// TIA Portal V17 export
// export: Created 2022-07-28T18:02:47.3020839Z, ExportSetting None, DisplayName Totally Integrated Automation Portal, DisplayVersion V17, DisplayName TIA Portal Openness, DisplayVersion V17, DisplayName TIA Portal Teamcenter Gateway, DisplayVersion V17, DisplayName TIA Portal Version Control Interface, DisplayVersion V17, DisplayName TIA Portal Test Suite Advanced, DisplayVersion V17, DisplayName SINAMICS Startdrive Advanced, DisplayVersion V17, DisplayName SINAMICS DCC, DisplayVersion V17, DisplayName SINAMICS Startdrive G130, G150, S120, S150, SINAMICS MV, S210, DisplayVersion V17, DisplayName SINAMICS Startdrive G110M, G120, G120C, G120D, G120P, G115D, DisplayVersion V17, DisplayName STEP 7 Professional, DisplayVersion V17, DisplayName SIMATIC Energy Suite, DisplayVersion V17, DisplayName STEP 7 CFC, DisplayVersion V17, DisplayName STEP 7 Safety, DisplayVersion V17, DisplayName WinCC Advanced / Unified PC, DisplayVersion V17, DisplayName SIMATIC Visualization Architect, DisplayVersion V17
FUNCTION_BLOCK "Internal_H05_FB"   // FB11, SCL
TITLE = InternalH01
{ S7_Optimized_Access := 'TRUE' }
// Proccess signals from fuses, safety and others internal devices
// stored: MemoryReserve 100, SetENOAutomatically false
   VAR_INPUT
      I_CmdGeneralReset { ExternalAccessible := 'False'; ExternalVisible := 'False'; ExternalWritable := 'False'} : Bool;   // 0 ⮥ 1 = Input general reset ERROR/Interlocks
      IR_CycleTime { ExternalAccessible := 'False'; ExternalVisible := 'False'; ExternalWritable := 'False'} : Real := 0.0;   // Time of last PLC cycle, sec
      I_Initialization { ExternalAccessible := 'False'; ExternalVisible := 'False'; ExternalWritable := 'False'} : Bool := FALSE;   // 1 = Restart PLC is active (First scan)
      I_One_1s { ExternalAccessible := 'False'; ExternalVisible := 'False'; ExternalWritable := 'False'} : Bool;   // 1 = One cycle per one seccond pulse
      I_Sup24_Ok { ExternalAccessible := 'False'; ExternalVisible := 'False'; ExternalWritable := 'False'} : Bool;   // 24 VDC OK 004 -T1
      I_UPS_Alarm_Ok { ExternalAccessible := 'False'; ExternalVisible := 'False'; ExternalWritable := 'False'} : Bool;   // БЛОК безперебійного електроживлення ALARM 004 -K1.1
      I_UPS_Bat_Ok { ExternalAccessible := 'False'; ExternalVisible := 'False'; ExternalWritable := 'False'} : Bool;   // БЛОК безперебійного електроживлення BAT. 004 -K1.2
      I_QF_DQ_Ok { ExternalAccessible := 'False'; ExternalVisible := 'False'; ExternalWritable := 'False'} : Bool;   // Живлення модулів DO 004 -F4
      I_QF_AI_Ok { ExternalAccessible := 'False'; ExternalVisible := 'False'; ExternalWritable := 'False'} : Bool;   // Живлення модулів АІ 004 -F5
      I_QF_AQ_Ok { ExternalAccessible := 'False'; ExternalVisible := 'False'; ExternalWritable := 'False'} : Bool;   // Живлення модулів АО 004 -F6
      I_QF_Desmet_IM_Ok { ExternalAccessible := 'False'; ExternalVisible := 'False'; ExternalWritable := 'False'} : Bool;   // Живлення ЕТ станції для контролера DESMET 004 -F7
      I_QF_Desmet_DI_DQ_Ok { ExternalAccessible := 'False'; ExternalVisible := 'False'; ExternalWritable := 'False'} : Bool;   // Жилвення модулів DI та DO для контролера DESMET 004 -F8
      I_QF_Desmet_AI_AQ_Ok { ExternalAccessible := 'False'; ExternalVisible := 'False'; ExternalWritable := 'False'} : Bool;   // Живлення модулів AI та АO для контролера DESMET 004 -F9
      I_QF_Inv_Ctrl_Ok { ExternalAccessible := 'False'; ExternalVisible := 'False'; ExternalWritable := 'False'} : Bool;   // Живлення модулів керування частотників 004 -F10
      I_QF_Inv_STO_Ok { ExternalAccessible := 'False'; ExternalVisible := 'False'; ExternalWritable := 'False'} : Bool;   // Живлення STO контактів, частотних перетворювачів 004 -F11
      I_QF_Internal_Ok { ExternalAccessible := 'False'; ExternalVisible := 'False'; ExternalWritable := 'False'} : Bool;   // Живлення внутрішніх кіл 004 -F12
      I_QF_SafRelay_Ok { ExternalAccessible := 'False'; ExternalVisible := 'False'; ExternalWritable := 'False'} : Bool;   // Живлення реле безпеки 004 -F13
      I_QF_Analog_Ok { ExternalAccessible := 'False'; ExternalVisible := 'False'; ExternalWritable := 'False'} : Bool;   // Живлення аналогових сигналів 004 -F14
      I_QF_ThermoRelay_Ok { ExternalAccessible := 'False'; ExternalVisible := 'False'; ExternalWritable := 'False'} : Bool;   // Живлення термореле 004 -F15
      I_QF_VlvDisFoam_Ok { ExternalAccessible := 'False'; ExternalVisible := 'False'; ExternalWritable := 'False'} : Bool;   // Живлення клапанів ємності антивспінювача 004 -F16
      I_QF_FlowMeters_Ok { ExternalAccessible := 'False'; ExternalVisible := 'False'; ExternalWritable := 'False'} : Bool;   // Живлення витратомірів 004 -F17
      I_QF_VlvVitamin_Ok { ExternalAccessible := 'False'; ExternalVisible := 'False'; ExternalWritable := 'False'} : Bool;   // Живлення клапанів ємності вітамінів 004 -F18
      I_QF_DI_DQ_1_Ok { ExternalAccessible := 'False'; ExternalVisible := 'False'; ExternalWritable := 'False'} : Bool;   // Живлення дискретних сигналів 004 -F19
      I_QF_DI_DQ_2_Ok { ExternalAccessible := 'False'; ExternalVisible := 'False'; ExternalWritable := 'False'} : Bool;   // Живлення дискретних сигналів 004 -F20
      I_QS_Scalance_Ok { ExternalAccessible := 'False'; ExternalVisible := 'False'; ExternalWritable := 'False'} : Bool;   // Живлення скаланса 004 -F21
      I_SB_ES_Box_Ok { ExternalAccessible := 'False'; ExternalVisible := 'False'; ExternalWritable := 'False'} : Bool;   // Аварійний стоп 005 -SB1
      I_SB_ES_Ack_Ok { ExternalAccessible := 'False'; ExternalVisible := 'False'; ExternalWritable := 'False'} : Bool;   // Квітування 005 -SB2
      I_KM_SafRelay_Ok { ExternalAccessible := 'False'; ExternalVisible := 'False'; ExternalWritable := 'False'} : Bool;   // Доп. котакти контакторів кіл безпеки 005 -KM2
   END_VAR
   VAR_OUTPUT
      QW_STW { ExternalWritable := 'False'} : Word;   // Status for HMI
      QW_MW1 { ExternalWritable := 'False'} : Word;   // Message word for HMI 1
      QW_MW2 { ExternalWritable := 'False'} : Word := 16#0;   // Message word for HMI 2
      QW_MW3 { ExternalWritable := 'False'} : Word := 16#0;   // Message word for HMI 3
      Q_Reset { ExternalAccessible := 'False'; ExternalVisible := 'False'; ExternalWritable := 'False'} : Bool;   // 1 = Reset external err
      Q_SomeErr { ExternalAccessible := 'False'; ExternalVisible := 'False'; ExternalWritable := 'False'} : Bool;   // 1 = Some err occured
      Q_Sup24_Ok { ExternalAccessible := 'False'; ExternalVisible := 'False'; ExternalWritable := 'False'} : Bool;   // 24 VDC OK 004 -T1
      Q_UPS_Alarm_Ok { ExternalAccessible := 'False'; ExternalVisible := 'False'; ExternalWritable := 'False'} : Bool;   // БЛОК безперебійного електроживлення ALARM 004 -K1.1
      Q_UPS_Bat_Ok { ExternalAccessible := 'False'; ExternalVisible := 'False'; ExternalWritable := 'False'} : Bool;   // БЛОК безперебійного електроживлення BAT. 004 -K1.2
      Q_QF_DQ_Ok { ExternalAccessible := 'False'; ExternalVisible := 'False'; ExternalWritable := 'False'} : Bool;   // Живлення модулів DO 004 -F4
      Q_QF_AI_Ok { ExternalAccessible := 'False'; ExternalVisible := 'False'; ExternalWritable := 'False'} : Bool;   // Живлення модулів АІ 004 -F5
      Q_QF_AQ_Ok { ExternalAccessible := 'False'; ExternalVisible := 'False'; ExternalWritable := 'False'} : Bool;   // Живлення модулів АО 004 -F6
      Q_QF_Desmet_IM_Ok { ExternalAccessible := 'False'; ExternalVisible := 'False'; ExternalWritable := 'False'} : Bool;   // Живлення ЕТ станції для контролера DESMET 004 -F7
      Q_QF_Desmet_DI_DQ_Ok { ExternalAccessible := 'False'; ExternalVisible := 'False'; ExternalWritable := 'False'} : Bool;   // Жилвення модулів DI та DO для контролера DESMET 004 -F8
      Q_QF_Desmet_AI_AQ_Ok { ExternalAccessible := 'False'; ExternalVisible := 'False'; ExternalWritable := 'False'} : Bool;   // Живлення модулів AI та АO для контролера DESMET 004 -F9
      Q_QF_Inv_Ctrl_Ok { ExternalAccessible := 'False'; ExternalVisible := 'False'; ExternalWritable := 'False'} : Bool;   // Живлення модулів керування частотників 004 -F10
      Q_QF_Inv_STO_Ok { ExternalAccessible := 'False'; ExternalVisible := 'False'; ExternalWritable := 'False'} : Bool;   // Живлення STO контактів, частотних перетворювачів 004 -F11
      Q_QF_Internal_Ok { ExternalAccessible := 'False'; ExternalVisible := 'False'; ExternalWritable := 'False'} : Bool;   // Живлення внутрішніх кіл 004 -F12
      Q_QF_SafRelay_Ok { ExternalAccessible := 'False'; ExternalVisible := 'False'; ExternalWritable := 'False'} : Bool;   // Живлення реле безпеки 004 -F13
      Q_QF_Analog_Ok { ExternalAccessible := 'False'; ExternalVisible := 'False'; ExternalWritable := 'False'} : Bool;   // Живлення аналогових сигналів 004 -F14
      Q_QF_ThermoRelay_Ok { ExternalAccessible := 'False'; ExternalVisible := 'False'; ExternalWritable := 'False'} : Bool;   // Живлення термореле 004 -F15
      Q_QF_VlvDisFoam_Ok { ExternalAccessible := 'False'; ExternalVisible := 'False'; ExternalWritable := 'False'} : Bool;   // Живлення клапанів ємності антивспінювача 004 -F16
      Q_QF_FlowMeters_Ok { ExternalAccessible := 'False'; ExternalVisible := 'False'; ExternalWritable := 'False'} : Bool;   // Живлення витратомірів 004 -F17
      Q_QF_VlvVitamin_Ok { ExternalAccessible := 'False'; ExternalVisible := 'False'; ExternalWritable := 'False'} : Bool;   // Живлення клапанів ємності вітамінів 004 -F18
      Q_QF_DI_DQ_1_Ok { ExternalAccessible := 'False'; ExternalVisible := 'False'; ExternalWritable := 'False'} : Bool;   // Живлення дискретних сигналів 004 -F19
      Q_QF_DI_DQ_2_Ok { ExternalAccessible := 'False'; ExternalVisible := 'False'; ExternalWritable := 'False'} : Bool;   // Живлення дискретних сигналів 004 -F20
      Q_QS_Scalance_Ok { ExternalAccessible := 'False'; ExternalVisible := 'False'; ExternalWritable := 'False'} : Bool;   // Живлення скаланса 004 -F21
      Q_KM_SafRelay_Ok { ExternalAccessible := 'False'; ExternalVisible := 'False'; ExternalWritable := 'False'} : Bool;   // Доп. котакти контакторів кіл безпеки 005 -KM2
   END_VAR
   VAR_IN_OUT
      II_CMD : Int;   // Command from HMI for current box
   END_VAR
   VAR
      s_Sup24_Err { ExternalAccessible := 'False'; ExternalVisible := 'False'; ExternalWritable := 'False'} : Bool;   // 24 VDC OK 004 -T1
      s_UPS_Alarm_Err { ExternalAccessible := 'False'; ExternalVisible := 'False'; ExternalWritable := 'False'} : Bool;   // БЛОК безперебійного електроживлення ALARM 004 -K1.1
      s_UPS_Bat_Err { ExternalAccessible := 'False'; ExternalVisible := 'False'; ExternalWritable := 'False'} : Bool;   // БЛОК безперебійного електроживлення BAT. 004 -K1.2
      s_QF_DQ_Err { ExternalAccessible := 'False'; ExternalVisible := 'False'; ExternalWritable := 'False'} : Bool;   // Живлення модулів DO 004 -F4
      s_QF_AI_Err { ExternalAccessible := 'False'; ExternalVisible := 'False'; ExternalWritable := 'False'} : Bool;   // Живлення модулів АІ 004 -F5
      s_QF_AQ_Err { ExternalAccessible := 'False'; ExternalVisible := 'False'; ExternalWritable := 'False'} : Bool;   // Живлення модулів АО 004 -F6
      s_QF_Desmet_IM_Err { ExternalAccessible := 'False'; ExternalVisible := 'False'; ExternalWritable := 'False'} : Bool;   // Живлення ЕТ станції для контролера DESMET 004 -F7
      s_QF_Desmet_DI_DQ_Err { ExternalAccessible := 'False'; ExternalVisible := 'False'; ExternalWritable := 'False'} : Bool;   // Жилвення модулів DI та DO для контролера DESMET 004 -F8
      s_QF_Desmet_AI_AQ_Err { ExternalAccessible := 'False'; ExternalVisible := 'False'; ExternalWritable := 'False'} : Bool;   // Живлення модулів AI та АO для контролера DESMET 004 -F9
      s_QF_Inv_Ctrl_Err { ExternalAccessible := 'False'; ExternalVisible := 'False'; ExternalWritable := 'False'} : Bool;   // Живлення модулів керування частотників 004 -F10
      s_QF_Inv_STO_Err { ExternalAccessible := 'False'; ExternalVisible := 'False'; ExternalWritable := 'False'} : Bool;   // Живлення STO контактів, частотних перетворювачів 004 -F11
      s_QF_Internal_Err { ExternalAccessible := 'False'; ExternalVisible := 'False'; ExternalWritable := 'False'} : Bool;   // Живлення внутрішніх кіл 004 -F12
      s_QF_SafRelay_Err { ExternalAccessible := 'False'; ExternalVisible := 'False'; ExternalWritable := 'False'} : Bool;   // Живлення реле безпеки 004 -F13
      s_QF_Analog_Err { ExternalAccessible := 'False'; ExternalVisible := 'False'; ExternalWritable := 'False'} : Bool;   // Живлення аналогових сигналів 004 -F14
      s_QF_ThermoRelay_Err { ExternalAccessible := 'False'; ExternalVisible := 'False'; ExternalWritable := 'False'} : Bool;   // Живлення термореле 004 -F15
      s_QF_VlvDisFoam_Err { ExternalAccessible := 'False'; ExternalVisible := 'False'; ExternalWritable := 'False'} : Bool;   // Живлення клапанів ємності антивспінювача 004 -F16
      s_QF_FlowMeters_Err { ExternalAccessible := 'False'; ExternalVisible := 'False'; ExternalWritable := 'False'} : Bool;   // Живлення витратомірів 004 -F17
      s_QF_VlvVitamin_Err { ExternalAccessible := 'False'; ExternalVisible := 'False'; ExternalWritable := 'False'} : Bool;   // Живлення клапанів ємності вітамінів 004 -F18
      s_QF_DI_DQ_1_Err { ExternalAccessible := 'False'; ExternalVisible := 'False'; ExternalWritable := 'False'} : Bool;   // Живлення дискретних сигналів 004 -F19
      s_QF_DI_DQ_2_Err { ExternalAccessible := 'False'; ExternalVisible := 'False'; ExternalWritable := 'False'} : Bool;   // Живлення дискретних сигналів 004 -F20
      s_QS_Scalance_Err { ExternalAccessible := 'False'; ExternalVisible := 'False'; ExternalWritable := 'False'} : Bool;   // Живлення скаланса 004 -F21
      s_KM_SafRelay_Err { ExternalAccessible := 'False'; ExternalVisible := 'False'; ExternalWritable := 'False'} : Bool;   // Доп. котакти контакторів кіл безпеки 005 -KM2
      s_TP_Reset { ExternalAccessible := 'False'; ExternalVisible := 'False'; ExternalWritable := 'False'} : "Lib_FB_Timer_TP_Simple";
   END_VAR
   VAR_TEMP
      t_ResetHMI : Bool;   // Reset from HMI
      t_ResetLogic : Bool;   // Reset for logic
      t_SomeErr : Bool;   // 1 = Some err occured
      ti_LogicCMD : Int;   // CMD for logic
      tw_STW : Word;   // Status for HMI
      tw_MW1 : Word;   // Message word for HMI 1
      tw_MW2 : Word;   // Message word for HMI 2
      tw_MW3 : Word;   // Message word for HMI 3
   END_VAR
BEGIN
   REGION Initialization
       IF #II_CMD <> 0
       THEN
           #ti_LogicCMD := #II_CMD;
           #II_CMD := 0;
       ELSE
           #ti_LogicCMD := 0;
       END_IF;

       #t_ResetHMI := false;
       #tw_STW := w#16#0;
       #tw_MW1 := w#16#0;
       #tw_MW2 := w#16#0;
       #tw_MW3 := w#16#0;
   END_REGION

   REGION Reset for logic
       //Reset from HMI
       CASE #ti_LogicCMD OF
           31..32:  //Reset
               #t_ResetHMI := true;
           ELSE  // Statement section ELSE
               ;
       END_CASE;

       //Reset for logic
       #t_ResetLogic := #t_ResetHMI
       OR #I_CmdGeneralReset
       OR #I_SB_ES_Ack_Ok;

       #s_TP_Reset(IR_CycleTime:=#IR_CycleTime,
                   IB_StartTimerInput:=#t_ResetLogic,
                   IR_SpTime:=2.0,
                   QB_TimerOut=>#t_ResetLogic);

   END_REGION

   REGION Catch errors
       #s_Sup24_Err := (NOT #I_Sup24_Ok
       OR (#s_Sup24_Err
       AND NOT #t_ResetLogic))
       AND NOT #I_Initialization;

       #s_UPS_Alarm_Err := (NOT #I_UPS_Alarm_Ok
       OR (#s_UPS_Alarm_Err
       AND NOT #t_ResetLogic))
       AND NOT #I_Initialization;

       #s_UPS_Bat_Err := (NOT #I_UPS_Bat_Ok
       OR (#s_UPS_Bat_Err
       AND NOT #t_ResetLogic))
       AND NOT #I_Initialization;

       #s_QF_DQ_Err := (NOT #I_QF_DQ_Ok
       OR (#s_QF_DQ_Err
       AND NOT #t_ResetLogic))
       AND NOT #I_Initialization;

       #s_QF_AI_Err := (NOT #I_QF_AI_Ok
       OR (#s_QF_AI_Err
       AND NOT #t_ResetLogic))
       AND NOT #I_Initialization;

       #s_QF_AQ_Err := (NOT #I_QF_AQ_Ok
       OR (#s_QF_AQ_Err
       AND NOT #t_ResetLogic))
       AND NOT #I_Initialization;

       #s_QF_Desmet_IM_Err := (NOT #I_QF_Desmet_IM_Ok
       OR (#s_QF_Desmet_IM_Err
       AND NOT #t_ResetLogic))
       AND NOT #I_Initialization;

       #s_QF_Desmet_DI_DQ_Err := (NOT #I_QF_Desmet_DI_DQ_Ok
       OR (#s_QF_Desmet_DI_DQ_Err
       AND NOT #t_ResetLogic))
       AND NOT #I_Initialization;

       #s_QF_Desmet_AI_AQ_Err := (NOT #I_QF_Desmet_AI_AQ_Ok
       OR (#s_QF_Desmet_AI_AQ_Err
       AND NOT #t_ResetLogic))
       AND NOT #I_Initialization;

       #s_QF_Inv_Ctrl_Err := (NOT #I_QF_Inv_Ctrl_Ok
       OR (#s_QF_Inv_Ctrl_Err
       AND NOT #t_ResetLogic))
       AND NOT #I_Initialization;

       #s_QF_Inv_STO_Err := (NOT #I_QF_Inv_STO_Ok
       OR (#s_QF_Inv_STO_Err
       AND NOT #t_ResetLogic))
       AND NOT #I_Initialization;

       #s_QF_Internal_Err := (NOT #I_QF_Internal_Ok
       OR (#s_QF_Internal_Err
       AND NOT #t_ResetLogic))
       AND NOT #I_Initialization;

       #s_QF_SafRelay_Err := (NOT #I_QF_SafRelay_Ok
       OR (#s_QF_SafRelay_Err
       AND NOT #t_ResetLogic))
       AND NOT #I_Initialization;

       #s_QF_Analog_Err := (NOT #I_QF_Analog_Ok
       OR (#s_QF_Analog_Err
       AND NOT #t_ResetLogic))
       AND NOT #I_Initialization;

       #s_QF_ThermoRelay_Err := (NOT #I_QF_ThermoRelay_Ok
       OR (#s_QF_ThermoRelay_Err
       AND NOT #t_ResetLogic))
       AND NOT #I_Initialization;

       #s_QF_VlvDisFoam_Err := (NOT #I_QF_VlvDisFoam_Ok
       OR (#s_QF_VlvDisFoam_Err
       AND NOT #t_ResetLogic))
       AND NOT #I_Initialization;

       #s_QF_FlowMeters_Err := (NOT #I_QF_FlowMeters_Ok
       OR (#s_QF_FlowMeters_Err
       AND NOT #t_ResetLogic))
       AND NOT #I_Initialization;

       #s_QF_VlvVitamin_Err := (NOT #I_QF_VlvVitamin_Ok
       OR (#s_QF_VlvVitamin_Err
       AND NOT #t_ResetLogic))
       AND NOT #I_Initialization;

       #s_QF_DI_DQ_1_Err := (NOT #I_QF_DI_DQ_1_Ok
       OR (#s_QF_DI_DQ_1_Err
       AND NOT #t_ResetLogic))
       AND NOT #I_Initialization;

       #s_QF_DI_DQ_2_Err := (NOT #I_QF_DI_DQ_2_Ok
       OR (#s_QF_DI_DQ_2_Err
       AND NOT #t_ResetLogic))
       AND NOT #I_Initialization;

       #s_QS_Scalance_Err := (NOT #I_QS_Scalance_Ok
       OR (#s_QS_Scalance_Err
       AND NOT #t_ResetLogic))
       AND NOT #I_Initialization;

       #s_KM_SafRelay_Err := (NOT #I_KM_SafRelay_Ok
       OR (#s_KM_SafRelay_Err
       AND NOT #t_ResetLogic
       AND NOT #I_SB_ES_Ack_Ok))
       AND NOT #I_Initialization;
   END_REGION

   REGION Write STW
       //Some err occured
       #t_SomeErr := #s_Sup24_Err
       OR #s_UPS_Alarm_Err
       OR #s_UPS_Bat_Err
       OR #s_QF_DQ_Err
       OR #s_QF_AI_Err
       OR #s_QF_AQ_Err
       OR #s_QF_Desmet_IM_Err
       OR #s_QF_Desmet_DI_DQ_Err
       OR #s_QF_Desmet_AI_AQ_Err
       OR #s_QF_Inv_Ctrl_Err
       OR #s_QF_Inv_STO_Err
       OR #s_QF_Internal_Err
       OR #s_QF_SafRelay_Err
       OR #s_QF_Analog_Err
       OR #s_QF_ThermoRelay_Err
       OR #s_QF_VlvDisFoam_Err
       OR #s_QF_FlowMeters_Err
       OR #s_QF_VlvVitamin_Err
       OR #s_QF_DI_DQ_1_Err
       OR #s_QF_DI_DQ_2_Err
       OR #s_QS_Scalance_Err
       OR #s_KM_SafRelay_Err;


       //Write err to STW
       #tw_STW.%X0 := #t_SomeErr;
       #tw_MW1.%X0 := #s_Sup24_Err;
       #tw_MW1.%X1 := #s_UPS_Alarm_Err;
       #tw_MW1.%X2 := #s_UPS_Bat_Err;
       #tw_MW1.%X3 := #s_QF_DQ_Err;
       #tw_MW1.%X4 := #s_QF_AI_Err;
       #tw_MW1.%X5 := #s_QF_AQ_Err;
       #tw_MW1.%X6 := #s_QF_Desmet_IM_Err;
       #tw_MW1.%X7 := #s_QF_Desmet_DI_DQ_Err;
       #tw_MW1.%X8 := #s_QF_Desmet_AI_AQ_Err;
       #tw_MW1.%X9 := #s_QF_Inv_Ctrl_Err;
       #tw_MW1.%X10 := #s_QF_Inv_STO_Err;
       #tw_MW1.%X11 := #s_QF_Internal_Err;
       #tw_MW1.%X12 := #s_QF_SafRelay_Err;
       #tw_MW1.%X13 := #s_QF_Analog_Err;
       #tw_MW1.%X14 := #s_QF_ThermoRelay_Err;
       #tw_MW2.%X0 := #s_QF_VlvDisFoam_Err;
       #tw_MW2.%X1 := #s_QF_FlowMeters_Err;
       #tw_MW2.%X2 := #s_QF_VlvVitamin_Err;
       #tw_MW2.%X3 := #s_QF_DI_DQ_1_Err;
       #tw_MW2.%X4 := #s_QF_DI_DQ_2_Err;
       #tw_MW2.%X5 := #s_QS_Scalance_Err;
       #tw_MW2.%X6 := #s_KM_SafRelay_Err;
   END_REGION

   REGION Write outs
       #QW_STW := #tw_STW;
       #Q_Reset := #t_ResetLogic;
       #Q_SomeErr := #t_SomeErr;
       #Q_Sup24_Ok := NOT #s_Sup24_Err;
       #Q_UPS_Alarm_Ok := NOT #s_UPS_Alarm_Err;
       #Q_UPS_Bat_Ok := NOT #s_UPS_Bat_Err;
       #Q_QF_DQ_Ok := NOT #s_QF_DQ_Err;
       #Q_QF_AI_Ok := NOT #s_QF_AI_Err;
       #Q_QF_AQ_Ok := NOT #s_QF_AQ_Err;
       #Q_QF_Desmet_IM_Ok := NOT #s_QF_Desmet_IM_Err;
       #Q_QF_Desmet_DI_DQ_Ok := NOT #s_QF_Desmet_DI_DQ_Err;
       #Q_QF_Desmet_AI_AQ_Ok := NOT #s_QF_Desmet_AI_AQ_Err;
       #Q_QF_Inv_Ctrl_Ok := NOT #s_QF_Inv_Ctrl_Err;
       #Q_QF_Inv_STO_Ok := NOT #s_QF_Inv_STO_Err;
       #Q_QF_Internal_Ok := NOT #s_QF_Internal_Err;
       #Q_QF_SafRelay_Ok := NOT #s_QF_SafRelay_Err;
       #Q_QF_Analog_Ok := NOT #s_QF_Analog_Err;
       #Q_QF_ThermoRelay_Ok := NOT #s_QF_ThermoRelay_Err;
       #Q_QF_VlvDisFoam_Ok := NOT #s_QF_VlvDisFoam_Err;
       #Q_QF_FlowMeters_Ok := NOT #s_QF_FlowMeters_Err;
       #Q_QF_VlvVitamin_Ok := NOT #s_QF_VlvVitamin_Err;
       #Q_QF_DI_DQ_1_Ok := NOT #s_QF_DI_DQ_1_Err;
       #Q_QF_DI_DQ_2_Ok := NOT #s_QF_DI_DQ_2_Err;
       #Q_QS_Scalance_Ok := NOT #s_QS_Scalance_Err;
       #Q_KM_SafRelay_Ok := NOT #s_KM_SafRelay_Err;
   END_REGION
END_FUNCTION_BLOCK
